{attribute 'qualified_only'}
{attribute 'strict'}
TYPE EN_TempControlMode_1 :
(
	TEMP_MODE_MANUAL := 1,
	TEMP_MODE_HEATCOOL,
	TEMP_MODE_STERI
);
END_TYPE

(* stored: Version 1.1.0.1, ProductVersion 3.1.4022.12
   DUT EN_TempControlMode_1: Id {1cdd0b24-858f-477d-aaf2-60002c7b414f} *)
